(* IEC 61131-3 sources: json/src/Elements, 3 files *)

(* ---- IJsonElement.st ---- *)
NAMESPACE Simatic.Ax.Json
    INTERFACE IJsonElement
        METHOD ToString : STRING
        END_METHOD

        METHOD Serialize : BOOL
            VAR_INPUT
                t : Array[*] OF BYTE;
            END_VAR
        END_METHOD
    END_INTERFACE
END_NAMESPACE

(* ---- IJsonElementMuteable.st ---- *)
NAMESPACE Simatic.Ax.Json
    INTERFACE IJsonElementMuteable
        METHOD HasNext : BOOL
        END_METHOD

        METHOD GetNext : IJsonElementMuteable
        END_METHOD

        METHOD AddElement
            VAR_INPUT
                elem : IJsonElement;
            END_VAR
        END_METHOD
    END_INTERFACE
END_NAMESPACE

(* ---- AbstractJsonElement.st ---- *)
USING System.Strings;
USING Simatic.Ax.Json;

NAMESPACE Simatic.Ax.Json
    CLASS ABSTRACT AbstractJsonElement IMPLEMENTS IJsonElementMuteable, IJsonElement
        VAR PUBLIC
            Key : STRING;
        END_VAR

        VAR PROTECTED
                _next : IJsonElementMuteable;
        END_VAR

        METHOD PUBLIC ABSTRACT ToString : STRING
        END_METHOD

        METHOD PUBLIC ABSTRACT Serialize : BOOL
            VAR_INPUT
                doc : REF_TO JsonDocument;
            END_VAR
        END_METHOD

        METHOD PROTECTED ToStringHelper : STRING
            VAR_INPUT
                valueAsString : STRING;
            END_VAR
            VAR_TEMP
                _str : STRING;
            END_VAR
            _str := Concat('"', Key, '"', ': "');
            _str := Concat(_str, valueAsString, '"');
            ToStringHelper := _str;
        END_METHOD

        METHOD PUBLIC SerializeHelper : DINT
            VAR_INPUT
                doc : REF_TO JsonDocument;
                valueAsString : STRING;
            END_VAR
            VAR_TEMP
                _i : DINT;
            END_VAR
            doc^.AddString(valueAsString);
        END_METHOD

        METHOD PUBLIC HasNext : BOOL
            HasNext := _next <> NULL;
        END_METHOD

        METHOD PUBLIC GetNext : IJsonElementMuteable
            GetNext := _next;
        END_METHOD

        METHOD PUBLIC Reset
            _next := NULL;
        END_METHOD

        METHOD PUBLIC Insert
            VAR_INPUT
                elem : IJsonElement;
            END_VAR
            IF _next = NULL THEN
                _next ?= elem;
            END_IF;
        END_METHOD

    END_CLASS
END_NAMESPACE
